/// Implicitly generated code : DO NOT EDIT!!!
/// checks for correct pointer use. Currently, this only detects null pointer, which are replaced by 
/// a pointer to a dummy area and reported as error
{attribute 'check_pointer' := ''}
{attribute 'no_check' := ''}
FUNCTION CheckPointer : POINTER TO BYTE
VAR_INPUT
	/// Destination address of the pointer
	ptToTest: POINTER TO BYTE;
	/// Size of the type the pointer points to. (e.g: 20 for POINTER TO ARRAY [0..9] OF INT) 
	iSize: DINT;
	/// Granularity of the pointer access. This is the size of the biggest non-structured data type in the type the pointer points to. (e.g: 2 for POINTER TO ARRAY [0..9] OF INT)
	iGran: DINT;
	/// Indicates read or write Access. TRUE = write access.
	bWrite: BOOL;
END_VAR

// check for outside address range
IF ptToTest = 0 THEN
	// report error 
	Services.fbEventHandler.Select(TC_Events.CodeEventClass.ErrorEvent)
						   .ArgSetString('pointer')
						   .Raise();
	// this is just a desparate way to keep the PLC from crashing, 
	// probably there's a better solution
	CheckPointer := ADR( MAIN ); 
END_IF

END_FUNCTION

(* stored: Version 1.1.0.1
   POU CheckPointer: Id {39657091-c17f-4b5b-beb4-1d0514bc4ef3}, SpecialFunc None *)
